// TIA Portal V20 export
// export: Created 2026-07-22T09:35:21.5663408Z, ExportSetting WithDefaults, DisplayName Totally Integrated Automation Portal, DisplayVersion V20, DisplayName TIA Portal Openness, DisplayVersion V20, DisplayName TIA Portal Version Control Interface, DisplayVersion V20, DisplayName STEP 7 Professional, DisplayVersion V20, DisplayName STEP 7 Safety, DisplayVersion V20, DisplayName WinCC Basic/Comfort/Advanced, DisplayVersion V20, DisplayName WinCC Professional, DisplayVersion V20, DisplayName WinCC Unified, DisplayVersion V20
ORGANIZATION_BLOCK "Main"   // OB1, LAD, ProgramCycle
TITLE = "Main Program Sweep (Cycle)"
{ S7_Optimized_Access := 'TRUE' }
VERSION : 0.1
// stored: AutoNumber true, IsIECCheckEnabled false, SetENOAutomatically false
   VAR_INPUT
      Initial_Call : Bool;   // Initial call of this OB
      Remanence : Bool;   // =True, if remanent data are available
   END_VAR
BEGIN

REGION Network 1
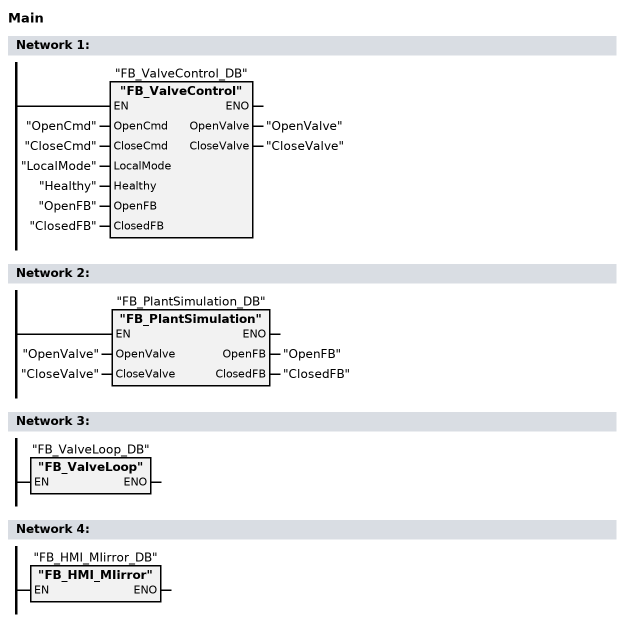
   RUNG wire#powerrail
      "FB_ValveControl_DB"(OpenCmd := "OpenCmd", CloseCmd := "CloseCmd", LocalMode := "LocalMode", Healthy := "Healthy", OpenFB := "OpenFB", ClosedFB := "ClosedFB", OpenValve => "OpenValve", CloseValve => "CloseValve")
   END_RUNG
   // the same network as SCL:
   "FB_ValveControl_DB"(OpenCmd := "OpenCmd",   // "FB_ValveControl"
                        CloseCmd := "CloseCmd",
                        LocalMode := "LocalMode",
                        Healthy := "Healthy",
                        OpenFB := "OpenFB",
                        ClosedFB := "ClosedFB",
                        OpenValve => "OpenValve",
                        CloseValve => "CloseValve");
END_REGION

REGION Network 2
   RUNG wire#powerrail
      "FB_PlantSimulation_DB"(OpenValve := "OpenValve", CloseValve := "CloseValve", OpenFB => "OpenFB", ClosedFB => "ClosedFB")
   END_RUNG
   // the same network as SCL:
   "FB_PlantSimulation_DB"(OpenValve := "OpenValve",   // "FB_PlantSimulation"
                           CloseValve := "CloseValve",
                           OpenFB => "OpenFB",
                           ClosedFB => "ClosedFB");
END_REGION

REGION Network 3
   RUNG wire#powerrail
      "FB_ValveLoop_DB"()
   END_RUNG
   // the same network as SCL:
   "FB_ValveLoop_DB"();   // "FB_ValveLoop"
END_REGION

REGION Network 4
   RUNG wire#powerrail
      "FB_HMI_MIirror_DB"()
   END_RUNG
   // the same network as SCL:
   "FB_HMI_MIirror_DB"();   // "FB_HMI_MIirror"
END_REGION
END_ORGANIZATION_BLOCK
